FUNCTION_BLOCK EcNetwork
VAR_INPUT
	enable : BOOL;
	netID : T_AmsNetId; //AmsNetID of the EtherCAT master node (NIC, EK1200, etc)
END_VAR
VAR_OUTPUT 
	slaves : ARRAY[0..EC_MAX_SLAVES] OF ST_EcSlaveConfigData; //devices
	slaveStates : ARRAY[0..EC_MAX_SLAVES] OF ST_EcSlaveState; //device states
	
	//start-end indexes for each subarea to access
	deviceIndexesA21 : ARRAY[0..1] OF DINT;
	deviceIndexesA22 : ARRAY[0..1] OF DINT;
	deviceIndexesA23 : ARRAY[0..1] OF DINT;
	deviceIndexesA24 : ARRAY[0..1] OF DINT;
	deviceIndexesA25 : ARRAY[0..1] OF DINT;
	deviceIndexesA26 : ARRAY[0..1] OF DINT;
END_VAR
VAR_OUTPUT
	numSlaves : DINT; //nSlaves must be cast from UINT to DINT in order to end iteration at -1 if there are no slaves
	
	diagnosticsError : BOOL;
	errorInit : BOOL;
	errorPreop : BOOL;
	errorBootstrap : BOOL;
	errorSafeop : BOOL;
	
	operational : BOOL;
END_VAR
VAR
	fbEcGetAllSlaveStates : FB_EcGetAllSlaveStates;
	fbEcGetConfiguredSlaves : FB_EcGetConfSlaves;
	
	i : DINT;
END_VAR

blocks();

diagnosticsError := fbEcGetAllSlaveStates.bError OR fbEcGetConfiguredSlaves.bError;
errorInit := FALSE;
errorPreop := FALSE;
errorBootstrap := FALSE;
errorSafeop := FALSE;

CheckEcNetwork(
	ecDeviceStates:= slaveStates, 
	ecIndex0:= 0, 
	ecIndex1:= numSlaves-1, 
	errorInit=> errorInit, 
	errorPreop=> errorPreop, 
	errorBootstrap=> errorBootstrap, 
	errorSafeop=> errorSafeop, 
	error=> , 
	operational=> operational);

distributeIndexes(slavePrefix:= 'A21', firstIndex=> deviceIndexesA21[0], lastIndex=> deviceIndexesA21[1]);
distributeIndexes(slavePrefix:= 'A22', firstIndex=> deviceIndexesA22[0], lastIndex=> deviceIndexesA22[1]);
distributeIndexes(slavePrefix:= 'A23', firstIndex=> deviceIndexesA23[0], lastIndex=> deviceIndexesA23[1]);
distributeIndexes(slavePrefix:= 'A24', firstIndex=> deviceIndexesA24[0], lastIndex=> deviceIndexesA24[1]);
distributeIndexes(slavePrefix:= 'A25', firstIndex=> deviceIndexesA25[0], lastIndex=> deviceIndexesA25[1]);
distributeIndexes(slavePrefix:= 'A26', firstIndex=> deviceIndexesA26[0], lastIndex=> deviceIndexesA26[1]);

METHOD PRIVATE blocks : BOOL
VAR_INST // added by the converter: edge detectors and wires of the graphical bodies
    _w1, _w2 : BOOL;
END_VAR
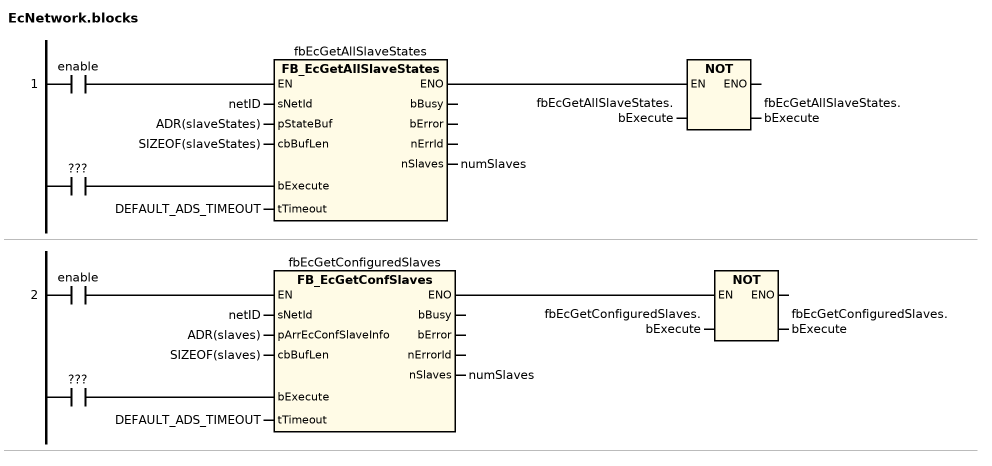
// NETWORK 1
_w1 := enable;
IF _w1 THEN
    fbEcGetAllSlaveStates(
        sNetId := netID,
        pStateBuf := ADR(slaveStates),
        cbBufLen := SIZEOF(slaveStates),
        tTimeout := DEFAULT_ADS_TIMEOUT,
        nSlaves => numSlaves); // FB_EcGetAllSlaveStates
END_IF
IF _w1 THEN fbEcGetAllSlaveStates.bExecute := NOT fbEcGetAllSlaveStates.bExecute; END_IF

// NETWORK 2
_w2 := enable;
IF _w2 THEN
    fbEcGetConfiguredSlaves(
        sNetId := netID,
        pArrEcConfSlaveInfo := ADR(slaves),
        cbBufLen := SIZEOF(slaves),
        tTimeout := DEFAULT_ADS_TIMEOUT,
        nSlaves => numSlaves); // FB_EcGetConfSlaves
END_IF
IF _w2 THEN fbEcGetConfiguredSlaves.bExecute := NOT fbEcGetConfiguredSlaves.bExecute; END_IF
END_METHOD

METHOD PRIVATE distributeIndexes : BOOL
VAR_INPUT
	slavePrefix : STRING;
END_VAR
VAR_OUTPUT
	firstIndex : DINT;
	lastIndex : DINT := -1; //no iteration if last index < first index
END_VAR
VAR
	firstIndexSet : BOOL;
	i : DINT;
END_VAR
FOR i:=0 TO numSlaves-1 BY 1 DO	
	IF NOT firstIndexSet THEN
		firstIndexSet := TRUE;
		firstIndex := i;
		
	ELSIF FIND(slaves[i].sName, slavePrefix) = 0 THEN
		RETURN;
		
	END_IF
	
	lastIndex := i;
	
END_FOR
END_METHOD

END_FUNCTION_BLOCK

(* stored: Version 1.1.0.1, ProductVersion 3.1.4024.11
   POU EcNetwork: Id {59e9e55a-f84d-4be9-a999-aeaebeda2db4}, SpecialFunc None
   Method blocks: Id {a89b65e8-9538-4fef-a0ab-eec6e9c813af}
   Method distributeIndexes: Id {e455c11b-54e8-41b1-b055-3837faecd446} *)
